(* CoDeSys 2.3.9.62 project: AperturaConClave.pro *)
(* Libraries: Standard.lib 2.6.14 11:37:46 *)

(* Global variable list: Global_Variables *)
VAR_GLOBAL

   (* Entradas *)
  (* Botonera de entrada *)
   Ent1:BOOL;
   Ent2:BOOL;
   Ent3:BOOL;
   Ent4:BOOL;
   Cierre:BOOL;


   (* Salidas *)
   CajaAbierta: BOOL;

   (*Claves *)
   Clave1:INT:=1;
  Clave2:INT:=2;
  Clave3:INT:=2;


END_VAR

(* POU PLC_PRG, ST *)
PROGRAM PLC_PRG
VAR
(*Necesitamos un tof*)
	Tempo:TOF;
	deco:INT:=0;
	estado:INT:=0;
	R1:R_TRIG; (* Seria más intuitivo un f-trig creo yo *)
	R2:R_TRIG;
	R3:R_TRIG;
	R4:R_TRIG;
	RC:R_TRIG;
END_VAR
Tempo(PT:=T#4s);
(* aqui realizo la decodificación*)
R1(CLK:= Ent1);
R2(CLK:= Ent2);
R3(CLK:= Ent3);
R4(CLK:= Ent4);
RC(CLK:= Cierre);
IF R1.Q  THEN
deco:= 1;
ELSIF R2.Q THEN
deco:= 2;
ELSIF R3.Q THEN
deco:= 3;
ELSIF R4.Q THEN
deco:= 4;
ELSE deco:= 0;
END_IF
(*Estados y su retorno *)
CASE estado OF
0:  IF deco = clave1 THEN
	estado:=1;
	END_IF;
	TEMPO.IN:= (deco = clave1);
1: IF deco = clave2 AND TEMPO.Q THEN
	estado:=2;
	ELSIF NOT TEMPO.Q OR   NOT( deco = 0 AND NOT( deco = clave1) ) THEN
	estado:=0;
	END_IF;
	TEMPO.IN := deco = clave2 AND TEMPO.Q;
2: IF deco = clave3 AND TEMPO.Q THEN
	estado:=3;
	ELSIF NOT TEMPO.Q OR   NOT( deco = 0 AND NOT( deco = clave2) ) THEN
	estado:=0;
	END_IF;
	TEMPO.IN := deco = clave3 AND TEMPO.Q;
3: IF RC.Q THEN
	estado:=0;
	CajaAbierta:= NOT RC.Q;
	ELSE CajaAbierta:= NOT RC.Q;
	END_IF;
	Tempo.IN:= FALSE;
ELSE estado:=0;
	Tempo.IN:= FALSE;
END_CASE;
END_PROGRAM

(* Visualisation Visu
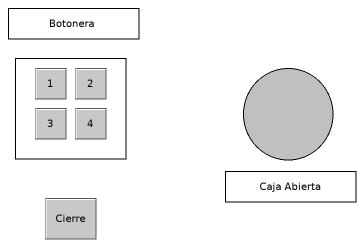
button at (50,130)-(81,161): text "1"; taps Ent1
button at (90,130)-(121,161): text "2"; taps Ent2
button at (50,170)-(81,201): text "3"; taps Ent3
button at (90,170)-(121,201): text "4"; taps Ent4
button at (60,260)-(111,301): text "Cierre"; taps Cierre
rectangle at (23,70)-(154,101): text "Botonera"
ellipse at (258,130)-(348,222): alarm colour if CajaAbierta
rectangle at (240,233)-(371,264): text "Caja Abierta"
1 more shapes without text or variables
*)
